// TwinCAT 3 PLC project Fraktal_Press_Demo
// Title: Fraktal_Press_Demo
// Company: fraktal-automation
// Author: fraktal-automation
// ProjectVersion: 0.1.0.10
// Description: CX2030 virtual/physical commissioning example: XTI-linked EK1200/EL1809/EL2809 HAL mapping, two-hand start, interlocked door/part slide, safety aliases, Control On/Off, AUTO/HOME/MANUAL, and model recipes.
// ProgramVersion: 3.1.4026.24
// libraries:
//   Fraktal_Core, 0.3.0.0 (fraktal-automation)
//   Fraktal_Modules, 0.2.0.0 (fraktal-automation)
//   Tc2_EtherCAT, * (Beckhoff Automation GmbH)
//   Tc2_Standard, * (Beckhoff Automation GmbH)
//   Tc2_System, * (Beckhoff Automation GmbH)
//   Tc3_Module, * (Beckhoff Automation GmbH)
// project tree:
//   00_System/Hardware/ GVL_PressIO.TcGVL (not stored), GVL_PressSafety.TcGVL (not stored)
//   00_System/ GVL_PressCommissioning.TcGVL, MAIN.TcPOU, FB_PressIoDriver.TcPOU (not stored), FB_PressControlOnCircuit.TcPOU, FB_PressControlDomain.TcPOU (not stored), FB_PressOutputAuthority.TcPOU (not stored), FB_PressSimulationDriver.TcPOU (not stored)
//   / PlcTask.TcTTO (not stored)
//   01_PneumaticPress/Sequences/ FB_PressDemoLoadPosition.TcPOU (not stored), FB_PressDemoHome.TcPOU (not stored), FB_PressDemoChangeover.TcPOU (not stored), FB_PressDemoAuto.TcPOU
//   01_PneumaticPress/Release/ FB_PressDemoRelease.TcPOU (not stored)
//   01_PneumaticPress/ FB_PressDemoUnit.TcPOU
//   01_PneumaticPress/Recipes/ FB_PressRecipeCatalog.TcPOU (not stored)
//   01_PneumaticPress/Io/ FB_PressIoCatalog.TcPOU (not stored), GVL_PressFieldbus.TcGVL (not stored)
// real-time tasks:
//   TASK PlcTask: cycle T#10ms, priority 20, ADS port 350
// I/O:
//   DEVICE =000+S-A610-A1 (EtherCAT)
// variable links:
//   Fraktal_Press_Demo/Fraktal_Press_Demo Instance <-> =000+S-A610-A1 (EtherCAT)/=000+S-K010 (EK1200)/=000+S-K010B1 (EL1809)
//     PlcTask Inputs/GVL_PressIO._000K910A <-> Channel 15/_000K910A
//     PlcTask Inputs/GVL_PressIO._000K911_Y32 <-> Channel 14/_000K911_Y32
//     PlcTask Inputs/GVL_PressIO._000MB085A_2 <-> Channel 10/_000MB085A_2
//     PlcTask Inputs/GVL_PressIO._000MB085A_4 <-> Channel 11/_000MB085A_4
//     PlcTask Inputs/GVL_PressIO._101B201A <-> Channel 3/_101B201A
//     PlcTask Inputs/GVL_PressIO._101B202A <-> Channel 5/_101B202A
//     PlcTask Inputs/GVL_PressIO._101B301A <-> Channel 1/_101B301A
//     PlcTask Inputs/GVL_PressIO._101B201B <-> Channel 4/_101B201B
//     PlcTask Inputs/GVL_PressIO._101B202B <-> Channel 6/_101B202B
//     PlcTask Inputs/GVL_PressIO._101B301B <-> Channel 2/_101B301B
//     PlcTask Inputs/GVL_PressIO._101B601 <-> Channel 12/_101B601
//     PlcTask Inputs/GVL_PressIO._101S101 <-> Channel 7/_101S101
//     PlcTask Inputs/GVL_PressIO._101S102 <-> Channel 8/_101S102
//   Fraktal_Press_Demo/Fraktal_Press_Demo Instance <-> =000+S-A610-A1 (EtherCAT)/=000+S-K010 (EK1200)/=000+S-K010C1 (EL2809)
//     PlcTask Outputs/GVL_PressIO._000K911_A1 <-> Channel 11/_000K911_A1
//     PlcTask Outputs/GVL_PressIO._000K951_A1 <-> Channel 10/_000K951_A1
//     PlcTask Outputs/GVL_PressIO._101K201A <-> Channel 3/_101K201A
//     PlcTask Outputs/GVL_PressIO._101K202A <-> Channel 5/_101K202A
//     PlcTask Outputs/GVL_PressIO._101K301A <-> Channel 1/_101K301A
//     PlcTask Outputs/GVL_PressIO._101K201B <-> Channel 4/_101K201B
//     PlcTask Outputs/GVL_PressIO._101K202B <-> Channel 6/_101K202B
//     PlcTask Outputs/GVL_PressIO._101K301B <-> Channel 2/_101K301B
//     PlcTask Outputs/GVL_PressIO._101P101 <-> Channel 7/_101P101
//     PlcTask Outputs/GVL_PressIO._101P102 <-> Channel 8/_101P102

// ---- 00_System/GVL_PressCommissioning.TcGVL
{attribute 'qualified_only'}
// Deployment-owned access-provider bootstrap. Secrets deliberately have no
// source default and are excluded from OPC UA; provision the retained values in
// the target's controlled commissioning workflow before locking the PLC policy.
VAR_GLOBAL PERSISTENT
    {attribute 'OPC.UA.DA' := '0'}
    OperatorPin   : STRING(32);
    {attribute 'OPC.UA.DA' := '0'}
    TechnicianPin : STRING(32);
    {attribute 'OPC.UA.DA' := '0'}
    AdminPin      : STRING(32);
END_VAR

// ---- 01_PneumaticPress/Sequences/FB_PressDemoAuto.TcPOU
// AUTO mode chain (Core §6.2/§6.8 ST skeleton on FB_SequenceBase): the continuous
// production cycle — await a fresh two-hand start with part+air present, transfer
// the part in, press for the recipe dwell, return to load position, count the good
// part, and loop until Stop. A Stop requested at the between-cycles wait is honored
// there (M_StopNow) so no phantom cycle is charged. Every child motion goes through
// the §6.1 handshake (M_MayIssue); progression rides the shared _retVal.
FUNCTION_BLOCK FB_PressDemoAuto EXTENDS FB_SequenceBase
VAR
    _partReady, _airReady, _startReady : BOOL;
    _dwellTwoHandHeld : BOOL;          // N220 named wait: two-hand held through the dwell
    _traceAccepted, _recordAccepted, _partProcessed : BOOL;
    {attribute 'OPC.UA.DA' := '0'}
    _pressRam : REFERENCE TO FB_CylinderCM;
    {attribute 'OPC.UA.DA' := '0'}
    _door : REFERENCE TO FB_CylinderCM;
    {attribute 'OPC.UA.DA' := '0'}
    _partSlide : REFERENCE TO FB_CylinderCM;
    {attribute 'OPC.UA.DA' := '0'}
    _twoHand : REFERENCE TO FB_TwoHandStartCM;
    {attribute 'OPC.UA.DA' := '0'}
    _partPresentSensor : REFERENCE TO FB_DigitalInputCM;
    {attribute 'OPC.UA.DA' := '0'}
    _airPressureMonitor : REFERENCE TO FB_AirPressureMonitorCM;
    {attribute 'OPC.UA.DA' := '0'}
    _parCfg : REFERENCE TO ST_PneumaticPressParCfg;
    {attribute 'OPC.UA.DA' := '0'}
    _outCmd : REFERENCE TO ST_PneumaticPressOutCmd;
    {attribute 'OPC.UA.DA' := '0'}
    _startLatched : REFERENCE TO BOOL;
    {attribute 'OPC.UA.DA' := '0'}
    _loadPosition : FB_PressDemoLoadPosition;
    _loadPositionRunning : BOOL;
END_VAR

METHOD M_Reset
M_ResetBase(0);
_loadPositionRunning := FALSE;
_loadPosition.M_Reset(BaseStepNo := 0);
END_METHOD

METHOD M_Run
IF NOT _attached THEN
    RETURN;
END_IF
CASE _step OF
    0:  // initialize
        M_Step(StepNo := 0, StepName := 'project.step.pressAutoInitialize',
            Awaits := 0, AwaitingLabel := '', TimeClass := E_TimeClass.WORK, ExpectedTime := T#0S);
        _outCmd.CycleCompleted := FALSE;
        _outCmd.Homed := FALSE;
        _outCmd.ChangeoverCompleted := FALSE;
        _loadPositionRunning := FALSE;
        _retVal := E_StepResult.ADVANCE;
        M_Advance(OnAdvance := 100, OnJump1 := -1, OnJump2 := -1, OnJump3 := -1);
    100:  // await a fresh two-hand start (the §8.11.1 cycle-start marker)
        M_Step(StepNo := 100, StepName := 'project.step.pressAwaitTwoHand',
            Awaits := 0, AwaitingLabel := '', TimeClass := E_TimeClass.WAIT_OPERATOR, ExpectedTime := T#0S);
        _outCmd.CycleCompleted := FALSE;
        _partReady := M_Await(Idx := 1, Label := 'project.condition.partPresent',
            Ok := _partPresentSensor.OutImm.Value AND _partPresentSensor.OutImm.Quality);
        _airReady := M_Await(Idx := 2, Label := 'project.condition.airPressureOk',
            Ok := _airPressureMonitor.OutImm.PressureOk);
        IF _parCfg.RequireTwoHandStart THEN
            _startReady := M_Await(Idx := 3, Label := 'project.condition.twoHandStart', Ok := _startLatched);
        ELSE
            _startReady := TRUE;
        END_IF
        IF M_StopPending() THEN
            M_StopNow();                       // stop accepted BETWEEN cycles: no phantom cycle
        ELSIF _partReady AND _airReady AND _startReady THEN
            _traceAccepted := M_PartReceived();
            _retVal := E_StepResult.ADVANCE;
        END_IF
        M_Advance(OnAdvance := 110, OnJump1 := -1, OnJump2 := -1, OnJump3 := -1);
    110:  // ram up
        M_Step(StepNo := 110, StepName := 'project.step.pressRamUp',
            Awaits := _pressRam, AwaitingLabel := 'PressRam.RETRACT', TimeClass := E_TimeClass.WORK, ExpectedTime := T#0S);
        IF M_MayIssue(Steppable := TRUE) THEN
            _pressRam.Abort := FALSE; _pressRam.Command := E_CylinderCommand.RETRACT; _pressRam.Execute := TRUE;
        END_IF
        IF _pressRam.Done THEN _pressRam.Execute := FALSE; _retVal := E_StepResult.ADVANCE; END_IF
        M_Advance(OnAdvance := 130, OnJump1 := -1, OnJump2 := -1, OnJump3 := -1);
    130:  // door open
        M_Step(StepNo := 130, StepName := 'project.step.pressDoorOpen',
            Awaits := _door, AwaitingLabel := 'Door.RETRACT', TimeClass := E_TimeClass.WORK, ExpectedTime := T#0S);
        IF M_MayIssue(Steppable := TRUE) THEN
            _door.Abort := FALSE; _door.Command := E_CylinderCommand.RETRACT; _door.Execute := TRUE;
        END_IF
        IF _door.Done THEN _door.Execute := FALSE; _retVal := E_StepResult.ADVANCE; END_IF
        M_Advance(OnAdvance := 150, OnJump1 := -1, OnJump2 := -1, OnJump3 := -1);
    150:  // slide inside (value-adding sequence begins)
        M_Step(StepNo := 150, StepName := 'project.step.pressSlideInside',
            Awaits := _partSlide, AwaitingLabel := 'PartSlide.EXTEND', TimeClass := E_TimeClass.WORK, ExpectedTime := T#0S);
        IF M_MayIssue(Steppable := TRUE) THEN
            M_PartStarted();
            _partSlide.Abort := FALSE; _partSlide.Command := E_CylinderCommand.EXTEND; _partSlide.Execute := TRUE;
        END_IF
        IF _partSlide.Done THEN _partSlide.Execute := FALSE; _retVal := E_StepResult.ADVANCE; END_IF
        M_Advance(OnAdvance := 170, OnJump1 := -1, OnJump2 := -1, OnJump3 := -1);
    170:  // transfer settle
        M_Step(StepNo := 170, StepName := 'project.step.pressTransferSettle',
            Awaits := 0, AwaitingLabel := '', TimeClass := E_TimeClass.WORK, ExpectedTime := _parCfg.TransferSettleTime);
        _retVal := M_Delay(PT := _parCfg.TransferSettleTime);
        M_Advance(OnAdvance := 180, OnJump1 := -1, OnJump2 := -1, OnJump3 := -1);
    180:  // door close
        M_Step(StepNo := 180, StepName := 'project.step.pressDoorClose',
            Awaits := _door, AwaitingLabel := 'Door.EXTEND', TimeClass := E_TimeClass.WORK, ExpectedTime := T#0S);
        IF M_MayIssue(Steppable := TRUE) THEN
            _door.Abort := FALSE; _door.Command := E_CylinderCommand.EXTEND; _door.Execute := TRUE;
        END_IF
        IF _door.Done THEN _door.Execute := FALSE; _retVal := E_StepResult.ADVANCE; END_IF
        M_Advance(OnAdvance := 200, OnJump1 := -1, OnJump2 := -1, OnJump3 := -1);
    200:  // ram down
        M_Step(StepNo := 200, StepName := 'project.step.pressRamDown',
            Awaits := _pressRam, AwaitingLabel := 'PressRam.EXTEND', TimeClass := E_TimeClass.WORK, ExpectedTime := T#0S);
        IF M_MayIssue(Steppable := TRUE) THEN
            _pressRam.Abort := FALSE; _pressRam.Command := E_CylinderCommand.EXTEND; _pressRam.Execute := TRUE;
        END_IF
        IF _pressRam.Done THEN _pressRam.Execute := FALSE; _retVal := E_StepResult.ADVANCE; END_IF
        M_Advance(OnAdvance := 220, OnJump1 := -1, OnJump2 := -1, OnJump3 := -1);
    220:  // press dwell — two-hand must stay held; releasing it HOLDS the dwell
        M_Step(StepNo := 220, StepName := 'project.step.pressDwell',
            Awaits := 0, AwaitingLabel := '', TimeClass := E_TimeClass.WORK, ExpectedTime := _parCfg.PressSettleTime);
        // Releasing the button mid-dwell is the designed way to stop pressing, so it
        // is a named wait (§6.9(b)), not a fault: the ram's outputs come off, the
        // dwell timer freezes where it is because M_Delay is not called, and pressing
        // again restores the force and finishes the remaining dwell. Faulting here
        // charged an unrecoverable downtime event for normal operator behaviour.
        _dwellTwoHandHeld := M_Await(Idx := 1, Label := 'project.condition.twoHandHeldDuringPress',
            Ok := _twoHand.OutImm.SafeActive OR NOT _parCfg.RequireTwoHandStart);
        IF NOT _dwellTwoHandHeld THEN
            _pressRam.WithdrawOutputs();
        ELSE
            // The press force is the valve latched by the EXTEND that step 200 already
            // completed, so after a withdraw only this call re-energizes it — and the
            // ram re-checks its own extend permit before it does (§7.2).
            _pressRam.RestoreOutputs();
            _retVal := M_Delay(PT := _parCfg.PressSettleTime);
        END_IF
        M_Advance(OnAdvance := 230, OnJump1 := -1, OnJump2 := -1, OnJump3 := -1);
    230:  // record the applied dwell (§3.16.1 measured value)
        M_Step(StepNo := 230, StepName := 'project.step.pressRecordResult',
            Awaits := 0, AwaitingLabel := '', TimeClass := E_TimeClass.WORK, ExpectedTime := T#0S);
        _recordAccepted := M_PartRecord(RecordName := 'PressDwell',
            Value := DINT_TO_LREAL(TIME_TO_DINT(_parCfg.PressSettleTime)),
            Minimum := 0, Maximum := 30000,
            Target := DINT_TO_LREAL(TIME_TO_DINT(_parCfg.PressSettleTime)), EngUnit := 'ms');
        _loadPositionRunning := FALSE;
        _retVal := E_StepResult.ADVANCE;
        M_Advance(OnAdvance := 240, OnJump1 := -1, OnJump2 := -1, OnJump3 := -1);
    240:  // return to the shared load-safe position (composite step)
        IF NOT _loadPositionRunning THEN
            _loadPosition.M_Reset(BaseStepNo := 240);
            _loadPositionRunning := TRUE;
        END_IF
        _loadPosition.M_Run();
        IF _loadPosition.Done THEN
            _loadPositionRunning := FALSE;
            _retVal := E_StepResult.ADVANCE;
        END_IF
        M_Advance(OnAdvance := 999, OnJump1 := -1, OnJump2 := -1, OnJump3 := -1);
    999:  // cycle complete — write result, count by verdict, loop (§8.11.1 finish marker)
        M_Step(StepNo := 999, StepName := 'project.step.pressAutoComplete',
            Awaits := 0, AwaitingLabel := '', TimeClass := E_TimeClass.WORK, ExpectedTime := T#0S);
        _outCmd.CycleCompleted := TRUE;
        _partProcessed := M_PartProcessed(Verdict := E_Verdict.OK, Reason := E_Reason.NONE);
        IF NOT _partProcessed THEN
            M_CountGood();                     // §3.9: no carrier configured — count directly
        END_IF
        _startLatched := FALSE;
        IF M_EndOfCycle() THEN
            _retVal := E_StepResult.ADVANCE;   // stop NOT requested: loop to N100
        END_IF
        M_Advance(OnAdvance := 100, OnJump1 := -1, OnJump2 := -1, OnJump3 := -1);
ELSE
    M_Fault(Reason := E_Reason.STEP_STALLED, DescriptionKey := 'std.error.undefinedStep');
END_CASE
END_METHOD

METHOD Setup : BOOL
VAR_INPUT
    Host : I_SequenceHost;
END_VAR
VAR_IN_OUT
    PressRam : FB_CylinderCM;
    Door : FB_CylinderCM;
    PartSlide : FB_CylinderCM;
    TwoHand : FB_TwoHandStartCM;
    PartPresentSensor : FB_DigitalInputCM;
    AirPressureMonitor : FB_AirPressureMonitorCM;
    ParCfg : ST_PneumaticPressParCfg;
    OutCmd : ST_PneumaticPressOutCmd;
    StartLatched : BOOL;
END_VAR
_pressRam REF= PressRam;
_door REF= Door;
_partSlide REF= PartSlide;
_twoHand REF= TwoHand;
_partPresentSensor REF= PartPresentSensor;
_airPressureMonitor REF= AirPressureMonitor;
_parCfg REF= ParCfg;
_outCmd REF= OutCmd;
_startLatched REF= StartLatched;
Setup := M_Attach(Host := Host) AND __ISVALIDREF(_pressRam) AND __ISVALIDREF(_door)
    AND __ISVALIDREF(_partSlide) AND __ISVALIDREF(_twoHand)
    AND __ISVALIDREF(_partPresentSensor) AND __ISVALIDREF(_airPressureMonitor)
    AND __ISVALIDREF(_parCfg) AND __ISVALIDREF(_outCmd) AND __ISVALIDREF(_startLatched)
    AND _loadPosition.Setup(Host := Host, PressRam := PressRam, Door := Door, PartSlide := PartSlide);
END_METHOD

END_FUNCTION_BLOCK

// ---- 01_PneumaticPress/FB_PressDemoUnit.TcPOU
// Project-owned Unit: pneumatic press + access door + transfer slide + two-hand request.
// Cylinder interlocks prevent the two documented collisions in AUTO and MANUAL.
// Certified E-stop, two-hand evaluation and safe valve outputs remain external.
FUNCTION_BLOCK FB_PressDemoUnit EXTENDS FB_UnitBase
VAR_INPUT
    ParCfg : ST_PneumaticPressParCfg;
    ParCmd : ST_PneumaticPressParCmd;
END_VAR
VAR_OUTPUT
    PressRam      : FB_CylinderCM;
    Door          : FB_CylinderCM;
    PartSlide     : FB_CylinderCM;
    TwoHand       : FB_TwoHandStartCM;
    PneumaticPower: FB_PowerGroupCM;
    PartPresentSensor : FB_DigitalInputCM;
    AirPressureMonitor : FB_AirPressureMonitorCM;
    ReleaseConditions : FB_PressDemoRelease; // project-owned, browseable condition state
    OutCmd        : ST_PneumaticPressOutCmd;
    OutImm        : ST_PneumaticPressOutImm;
END_VAR
VAR
    {attribute 'OPC.UA.DA' := '0'}
    _recipe : I_RecipeProvider;
    _parCfgStaged : ST_PneumaticPressParCfg;
    _recipePrepared : BOOL;
    _startLatched : BOOL;
    _powerRequestPending : BOOL;
    _powerTargetOn : BOOL;
    {attribute 'OPC.UA.DA' := '0'}
    _homeSequence : FB_PressDemoHome;       // §6.8 ST chain on FB_SequenceBase owns HOME steps
    {attribute 'OPC.UA.DA' := '0'}
    _changeoverSequence : FB_PressDemoChangeover;
    {attribute 'OPC.UA.DA' := '0'}
    _autoSequence : FB_PressDemoAuto;
END_VAR

Cyclic();

METHOD Setup : BOOL
VAR_INPUT
    Name : STRING(80);
    PressHal : REFERENCE TO ST_CylinderHal;
    DoorHal : REFERENCE TO ST_CylinderHal;
    SlideHal : REFERENCE TO ST_CylinderHal;
    TwoHandHal : REFERENCE TO ST_TwoHandHal;
    PowerHal : REFERENCE TO ST_PowerGroupHal;
    PartPresentHal : REFERENCE TO ST_DigitalInputHal;
    AirPressureHal : REFERENCE TO ST_AirPressureHal;
    Recipe : I_RecipeProvider;
END_VAR
VAR
    InitialModel : ST_ModelId;
    Ok : BOOL;
END_VAR
_M_SetName(Name);
_M_SetPresentation(DisplayNameKey := 'project.module.pneumaticPress.name', DescriptionKey := 'project.module.pneumaticPress.description');
_recipe := Recipe;
Ok := PressRam.Setup(Name := CONCAT(Name, '.PressRam'), HalRef := PressHal, Recipe := 0);
Ok := Door.Setup(Name := CONCAT(Name, '.Door'), HalRef := DoorHal, Recipe := 0) AND Ok;
Ok := PartSlide.Setup(Name := CONCAT(Name, '.PartSlide'), HalRef := SlideHal, Recipe := 0) AND Ok;
Ok := TwoHand.Setup(Name := CONCAT(Name, '.TwoHand'), HalRef := TwoHandHal) AND Ok;
Ok := PneumaticPower.Setup(Name := CONCAT(Name, '.PneumaticPower'), HalRef := PowerHal) AND Ok;
Ok := PartPresentSensor.Setup(Name := CONCAT(Name, '.PartPresentSensor'),
    HalRef := PartPresentHal, DisplayNameKey := 'project.module.partPresentSensor.name',
    DescriptionKey := 'project.module.partPresentSensor.description') AND Ok;
Ok := AirPressureMonitor.Setup(Name := CONCAT(Name, '.AirPressureMonitor'),
    HalRef := AirPressureHal) AND Ok;
Ok := ReleaseConditions.Setup(UnitPath := Name) AND Ok;
Ok := _homeSequence.Setup(Host := THIS^, PressRam := PressRam, Door := Door,
    PartSlide := PartSlide, OutCmd := OutCmd) AND Ok;
Ok := _changeoverSequence.Setup(Host := THIS^, PressRam := PressRam, Door := Door,
    PartSlide := PartSlide, OutCmd := OutCmd, Model := Model) AND Ok;
Ok := _autoSequence.Setup(Host := THIS^, PressRam := PressRam, Door := Door,
    PartSlide := PartSlide, TwoHand := TwoHand, PartPresentSensor := PartPresentSensor,
    AirPressureMonitor := AirPressureMonitor, ParCfg := ParCfg, OutCmd := OutCmd,
    StartLatched := _startLatched) AND Ok;
PneumaticPower.ParCfg.Kind := E_PowerGroupKind.VALVE_ZONE;
PneumaticPower.ParCfg.RequiredForControl := TRUE;
PneumaticPower.ParCfg.FieldbusLossReaction := E_FieldbusLossReaction.CONTROL_OFF;
Ok := _M_Register(PressRam) AND Ok;
Ok := _M_Register(Door) AND Ok;
Ok := _M_Register(PartSlide) AND Ok;
Ok := _M_Register(TwoHand) AND Ok;
Ok := _M_Register(PneumaticPower) AND Ok;
Ok := _M_Register(PartPresentSensor) AND Ok;
Ok := _M_Register(AirPressureMonitor) AND Ok;
Setup := Ok AND PrepareRecipe(Model := InitialModel);
IF Setup THEN CommitRecipe(); END_IF
END_METHOD

METHOD PrepareRecipe : BOOL
VAR_INPUT
    Model : ST_ModelId;
END_VAR
IF _recipe = 0 THEN
    _parCfgStaged := ParCfg;
    _recipePrepared := TRUE;
ELSIF _recipe.Load(ModelCode := Model.ModelCode, RecipeKey := 'PneumaticPressUnit', pParCfg := ADR(_parCfgStaged), Size := SIZEOF(_parCfgStaged)) THEN
    IF (_parCfgStaged.PressSettleTime > T#30S) OR (_parCfgStaged.TransferSettleTime > T#5S) THEN
        _M_Fault(E_Reason.RECIPE_INVALID, 'project.error.pressRecipeInvalid');
        _recipePrepared := FALSE;
        PrepareRecipe := FALSE;
        RETURN;
    END_IF
    _recipePrepared := TRUE;
ELSE
    _M_Fault(E_Reason.RECIPE_INVALID, 'std.error.recipeSchemaInvalid');
    _recipePrepared := FALSE;
    PrepareRecipe := FALSE;
    RETURN;
END_IF
PrepareRecipe := SUPER^.PrepareRecipe(Model := Model);
IF NOT PrepareRecipe THEN _recipePrepared := FALSE; END_IF
END_METHOD

METHOD CommitRecipe
SUPER^.CommitRecipe();
IF _recipePrepared THEN
    ParCfg := _parCfgStaged;
    // §8.11 performance references follow the model: OEE Performance denominator
    // and the WORK-time degradation baseline are per-recipe engineering data.
    Oee.IdealCycleMs := ParCfg.IdealCycleMs;
    Profiler.M_SetBaselineWork(WorkMs := ParCfg.BaselineWorkMs);
END_IF
_recipePrepared := FALSE;
END_METHOD

METHOD AbortRecipe
SUPER^.AbortRecipe();
_recipePrepared := FALSE;
END_METHOD

// First operational scan: initialize application-owned mode-chain state.
METHOD PROTECTED OnInit : DINT
OnInit := SUPER^.OnInit();
_M_ResetModeSequences();
_M_ClearModeTransitionState();
END_METHOD

// Every accepted Unit Start gets a fresh mode chain, including a repeated
// HOME/CHANGEOVER run that does not pass through another mode change.
METHOD PROTECTED OnCommandStart : DINT
OnCommandStart := SUPER^.OnCommandStart();
_M_ResetModeSequences();
END_METHOD

// Mode-entry wiring only. Step behavior remains in the selected sequence POU.
METHOD PROTECTED OnModeChanged : DINT
VAR_INPUT
    NewMode : E_Mode;
    OldMode : E_Mode;
END_VAR
OnModeChanged := SUPER^.OnModeChanged(
    NewMode := NewMode, OldMode := OldMode);
_M_ResetModeSequences();
_M_ClearModeTransitionState();
END_METHOD

METHOD PROTECTED OnCyclic : DINT
OnCyclic := SUPER^.OnCyclic();
// Project release engineering is a separate visible component. It owns the
// functional collision permits and mode-entry conditions consumed below.
ReleaseConditions.M_Evaluate(PressRam := PressRam, Door := Door, PartSlide := PartSlide,
    TwoHand := TwoHand, PneumaticPower := PneumaticPower,
    AirPressure := AirPressureMonitor);

// Latch access-gated Unit requests, then observe one full Execute-low scan before
// starting another power-group command (PLCopen edge discipline).
IF ControlOffRequest THEN
    _powerTargetOn := FALSE;
    _powerRequestPending := TRUE;
ELSIF ControlOnRequest THEN
    _powerTargetOn := TRUE;
    _powerRequestPending := TRUE;
END_IF
IF PneumaticPower.Done OR PneumaticPower.Error OR PneumaticPower.Aborted THEN
    PneumaticPower.Execute := FALSE;
ELSIF _powerRequestPending AND NOT PneumaticPower.Execute
AND (PneumaticPower.State = E_ExecState.READY) THEN
    PneumaticPower.Abort := FALSE;
    IF _powerTargetOn THEN
        PneumaticPower.Command := E_PowerGroupCommand.POWER_ON;
    ELSE
        PneumaticPower.Command := E_PowerGroupCommand.POWER_OFF;
    END_IF
    PneumaticPower.Execute := TRUE;
    _powerRequestPending := FALSE;
END_IF

// A physical two-hand edge may start AUTO from READY, or release an already
// running Unit's wait step. It never bypasses domain readiness or access policy.
IF TwoHand.OutImm.StartPulse
AND PartPresentSensor.OutImm.Value AND PartPresentSensor.OutImm.Quality
AND AirPressureMonitor.OutImm.PressureOk THEN
    IF (State = E_ExecState.BUSY) AND (ModeActive = E_Mode.AUTO) THEN
        _startLatched := TRUE;
    ELSIF (ModeActive = E_Mode.AUTO) AND Start() THEN
        _startLatched := TRUE;
    END_IF
ELSIF TwoHand.OutImm.StartPulse THEN
    _startLatched := FALSE;
END_IF
IF PneumaticPower.Error AND (State = E_ExecState.BUSY) THEN
    _M_RollupFault();
END_IF
IF (State = E_ExecState.BUSY)
AND NOT AirPressureMonitor.OutImm.PressureOk THEN
    PressRam.WithdrawOutputs();
    Door.WithdrawOutputs();
    PartSlide.WithdrawOutputs();
    _M_Fault(E_Reason.PERMISSIVE_NOT_MET, 'project.error.pressAirPressureLost');
END_IF
OutImm.PressRetracted := PressRam.OutImm.Retracted;
OutImm.DoorOpen := Door.OutImm.Retracted;
OutImm.DoorClosed := Door.OutImm.Extended;
OutImm.SlideInside := PartSlide.OutImm.Extended;
OutImm.SlideOutside := PartSlide.OutImm.Retracted;
OutImm.TwoHandArmed := TwoHand.OutImm.Armed;
OutImm.TwoHandActive := TwoHand.OutImm.SafeActive;
OutImm.PartPresent := PartPresentSensor.OutImm.Value AND PartPresentSensor.OutImm.Quality;
OutImm.AirPressureOk := AirPressureMonitor.OutImm.PressureOk;
OutImm.ReadyForLoad := Door.OutImm.Retracted AND NOT Door.OutImm.Extended
    AND PartSlide.OutImm.Retracted AND NOT PartSlide.OutImm.Extended
    AND PressRam.OutImm.Retracted AND NOT PressRam.OutImm.Extended;
OutImm.ActiveSettleTime := ParCfg.PressSettleTime;
OutImm.Diagnostic := Status.Diagnostic;
END_METHOD

METHOD PROTECTED OnAbort : DINT
OnAbort := SUPER^.OnAbort();
_M_PartAborted();                    // §3.16.3: the part leaves without a valid result
_M_WithdrawSequenceOutputs();
_M_ResetModeSequences();
_M_ClearModeTransitionState();
_powerTargetOn := FALSE;
_powerRequestPending := TRUE;
END_METHOD

// Error-state Abort is a deliberate recovery action but does not clear ERROR.
METHOD PROTECTED OnAbortInError : DINT
OnAbortInError := SUPER^.OnAbortInError();
_M_WithdrawSequenceOutputs();
_M_ResetModeSequences();
_M_ClearModeTransitionState();
_powerTargetOn := FALSE;
_powerRequestPending := TRUE;
END_METHOD

// An operator reset is recovering this Unit: put the application back to the same
// safe wiring an error-state abort establishes, so the reset the operator presses at
// the panel needs no separate Stop/Abort first. The base then releases the run
// command and the children's commands, so the next HOME gets a genuine command edge.
// Unlike the abort paths this does NOT touch control power in either direction: it
// never requests Control On (§9.8 forbids self-resume), and it must not request
// Control Off either — powering down a healthy control circuit would make the
// operator re-enable it before HOME could run, i.e. reintroduce the multi-action
// recovery this reset exists to remove. Power stays where the operator put it.
METHOD PROTECTED OnOperatorReset : DINT
OnOperatorReset := SUPER^.OnOperatorReset();
_M_WithdrawSequenceOutputs();
_M_ResetModeSequences();
_M_ClearModeTransitionState();
END_METHOD

// One safe-stop wiring point shared by normal and error-state abort transitions.
METHOD PROTECTED _M_WithdrawSequenceOutputs
PressRam.WithdrawOutputs();
Door.WithdrawOutputs();
PartSlide.WithdrawOutputs();
PressRam.Execute := FALSE;
Door.Execute := FALSE;
PartSlide.Execute := FALSE;
END_METHOD

// Reset application-owned chain plumbing at lifecycle transitions. The chains'
// N000/N999 steps remain the only owners of process initialization/completion.
METHOD PROTECTED _M_ResetModeSequences
_homeSequence.M_Reset();
_changeoverSequence.M_Reset();
_autoSequence.M_Reset();
END_METHOD

// Clear state that must not survive init, mode entry, or either abort path.
// OnCommandStart deliberately does not call this: a physical start pulse may have
// been latched one scan before the inherited Execute edge is consumed.
METHOD PROTECTED _M_ClearModeTransitionState
Decision.Prompt := '';
DecisionAnswer := 0;
_startLatched := FALSE;
END_METHOD

// Application-only seam for ordinary hardwired Control On/Off buttons.
// It is a method (not OPC UA data), so HMI writes still use the access-gated
// ReqControlOn/ReqControlOff contract. The power CM rechecks safety and health.
METHOD RequestLocalControl : BOOL
VAR_INPUT
    ControlOn : BOOL;
END_VAR
_powerTargetOn := ControlOn;
_powerRequestPending := TRUE;
RequestLocalControl := TRUE;
END_METHOD

// §3.4.2 — the press paces every motion boundary through _M_StepGate, so
// SINGLE_STEP and HOLD_TO_RUN are supported (NON-SAFETY pacing; interlocks
// and the certified safety layer are unaffected).
METHOD PROTECTED _M_SupportsRunStyle : BOOL
VAR_INPUT
    Style : E_RunStyle;
END_VAR
_M_SupportsRunStyle := (Style = E_RunStyle.CONTINUOUS)
    OR (Style = E_RunStyle.SINGLE_STEP) OR (Style = E_RunStyle.HOLD_TO_RUN);
END_METHOD

METHOD PROTECTED _M_Supports : BOOL
VAR_INPUT
    Mode : E_Mode;
END_VAR
_M_Supports := (Mode = E_Mode.AUTO) OR (Mode = E_Mode.MANUAL)
    OR (Mode = E_Mode.HOME) OR (Mode = E_Mode.CHANGEOVER);
END_METHOD

// Thin mode router. Each supported sequence is a named method in the Unit tree.
METHOD PROTECTED _M_Dispatch
CASE ModeActive OF
    E_Mode.AUTO:
        _M_SequenceAuto();
    E_Mode.HOME:
        _M_SequenceHome();
    E_Mode.CHANGEOVER:
        _M_SequenceChangeover();
    E_Mode.MANUAL:
        _M_Fault(E_Reason.UNSUPPORTED_COMMAND, 'project.error.pressManualHasNoSequence');
ELSE
    _M_Fault(E_Reason.UNSUPPORTED_COMMAND, 'project.error.pressModeHasNoSequence');
END_CASE
END_METHOD

// Wiring-only HOME adapter. OnCommandStart owns the reset edge; the sequence POU
// owns every process step and terminal action.
METHOD PROTECTED _M_SequenceHome
_homeSequence.M_Run();
END_METHOD

// Wiring-only CHANGEOVER adapter. The §6.8 chain owns model validation, safe
// positioning, the operator decision, and completion logic.
METHOD PROTECTED _M_SequenceChangeover
_changeoverSequence.M_Run();
END_METHOD

// Wiring-only AUTO adapter. Every production command, wait, timer, decision,
// traceability action, and transition lives in the §6.8 chain.
METHOD PROTECTED _M_SequenceAuto
_autoSequence.M_Run();
END_METHOD

METHOD PROTECTED _M_RouteManual : BOOL
VAR_INPUT
    TargetPath : STRING(255);
    Value : DINT;
END_VAR
_M_RouteManual := FALSE;
IF TargetPath = PressRam.Name THEN
    _M_RouteManual := PressRam.ManualCommand(Value := Value);
ELSIF TargetPath = Door.Name THEN
    _M_RouteManual := Door.ManualCommand(Value := Value);
ELSIF TargetPath = PartSlide.Name THEN
    _M_RouteManual := PartSlide.ManualCommand(Value := Value);
ELSE
    _M_RouteManual := FALSE;
END_IF
END_METHOD

// §7.8 mode-entry release owned by this Unit. The base Start method consumes the
// same report the HMI displays, so this condition cannot become explanation-only.
METHOD PROTECTED _M_AppendInterlocks
VAR_IN_OUT
    Report : ST_ReleaseReport;
END_VAR
ReleaseConditions.M_AppendStart(Report := Report);
END_METHOD

METHOD PROTECTED _M_AppendManualInterlocks
VAR_INPUT
    TargetPath : STRING(255);
    Value : DINT;
END_VAR
VAR_IN_OUT
    Report : ST_ReleaseReport;
END_VAR
ReleaseConditions.M_AppendManual(TargetPath := TargetPath, Value := Value,
    PressRam := PressRam, Door := Door, PartSlide := PartSlide, Report := Report);
END_METHOD

METHOD PROTECTED _M_PublishStatus
SUPER^._M_PublishStatus();
OutImm.Diagnostic := Status.Diagnostic;
END_METHOD

// §3.10.2 — base walk (Unit facets + all child modules), then the project-owned
// fieldbus topology identity: static members of GVL_PressFieldbus.Topology are
// OPC.UA.DA=0 and reach the HMI only through this manifest.
METHOD M_AppendConfig : BOOL
VAR_INPUT
    Pager : REFERENCE TO FB_ConfigPager;
END_VAR
M_AppendConfig := SUPER^.M_AppendConfig(Pager := Pager);
F_AppendTopologyConfig(Topology := GVL_PressFieldbus.Topology, Pager := Pager);
END_METHOD

END_FUNCTION_BLOCK

// ---- 00_System/MAIN.TcPOU
// Virtual-commissioning application for one pneumatic press Unit.
// IMPORTANT: the Safe* values below simulate TwinSAFE outputs only. A deployed
// machine maps certified E-stop/two-hand/guard/safe-valve results from TwinSAFE.
PROGRAM MAIN
VAR
    RecipeCatalog : FB_PressRecipeCatalog;
    PartCarrier : FB_LocalPartCarrier;    // §3.16.2 BY_POSITION identity + local result ring
    AccessUsers : FB_LocalAccessProvider; // §7.7 commissioning user/PIN table
    // TF6100 TMC-Filtered publication starts at the deployed root instance.
    // The marker is inherited by PneumaticPress's published child symbols.
    {attribute 'OPC.UA.DA' := '1'}
    PneumaticPress : FB_PressDemoUnit;
    IoCatalog : FB_PressIoCatalog;
    IoDriver : FB_PressIoDriver;
    ControlDomain : FB_PressControlDomain;
    OutputAuthority : FB_PressOutputAuthority;
    SimulationDriver : FB_PressSimulationDriver;
    PressHal, DoorHal, SlideHal : ST_CylinderHal;
    TwoHandHal : ST_TwoHandHal;
    PowerHal : ST_PowerGroupHal;
    PartPresentHal : ST_DigitalInputHal;
    AirPressureHal : ST_AirPressureHal;
    HealthProbe : FB_TcSystemHealthProbe;
    HealthConfig : ST_SystemHealthParCfg;
    HealthCpuLoadPct : LREAL;
    HealthMemoryAvailableMb : UDINT;
    HealthTimeSource : STRING(32);
    InitialModel : ST_ModelId;
    Plate : ST_Nameplate;
    Init : BOOL;
    // Read-only MIRRORS of the commissioning gates (see the VAR CONSTANT block).
    // They exist only so the gate state stays visible over ADS/OPC UA: the
    // compiler inlines constants, which may publish no symbol at all, and losing
    // that visibility would remove the fastest way to diagnose "no output moves".
    // They are reassigned from the constants every cycle and nothing reads them,
    // so writing one online is inert - the constant remains the only authority.
    UseSimulation : BOOL;
    ControlCircuitMappingConfirmed : BOOL;
    // §10.5.1 demand gate, written by the HMI while its fieldbus page is open.
    // FALSE parks the EtherCAT master scan (no ADS traffic for a view nobody is
    // watching); the last read states are held, never falsified.
    FieldbusViewActive : BOOL;

    // Simulation controls. E-stop is normally closed: TRUE = healthy circuit.
    SimEStopNc : BOOL := TRUE;
    SimControlOnButton : BOOL;
    SimControlOffButton : BOOL;
    SimLeftButton : BOOL;
    SimRightButton : BOOL;
    SimSafetyValveOk : BOOL := TRUE;
    SimFieldbusHealthy : BOOL := TRUE;
    SimPartPresent : BOOL := TRUE;
    SimAirPressureOk : BOOL := TRUE;
    SafeEStopOk : BOOL;
    SafeGuardClosed : BOOL;
    SafeTwoHandActive : BOOL;
    SafePneumaticPermit : BOOL;
    SafetyFieldbusHealthy : BOOL;
    StandardIoHealthy : BOOL;
    RawEStopHealthy : BOOL;
    LampsOn : BOOL;
    ControlOnEdge : R_TRIG;
    ControlOffEdge : R_TRIG;
    ControlOnAdopted : R_TRIG;   // rising edge of the relay chain's feedback
END_VAR
VAR CONSTANT
    // COMMISSIONING GATES - deliberately CONSTANT so they cannot be flipped
    // online. Defeating a gate must be a source change plus a download: a
    // reviewable, auditable act, not a live write from an HMI or ADS client.
    //
    // TRUE makes MAIN call M_ClearOutputs() every cycle, so no physical output
    // is ever energized while the simulation driver animates the plant.
    USE_SIMULATION : BOOL := FALSE;
    // FALSE makes M_WriteOutputs force _000K951_A1 and _000K911_A1 FALSE every
    // cycle. Control On then cannot energize, the hardwired N54 D2 relay chain
    // never closes, and NOTHING moves - even though the cylinder coils are
    // written unconditionally. Set TRUE only after verifying the K951/K911
    // electrical semantics on the cabinet; per N54 D2 SwitchControlOn and
    // EnableControlOn are distinct signals.
    CONTROL_CIRCUIT_MAPPING_CONFIRMED : BOOL := TRUE;
END_VAR

// Mirror the compile-time gates so they remain observable (see declaration).
UseSimulation := USE_SIMULATION;
ControlCircuitMappingConfirmed := CONTROL_CIRCUIT_MAPPING_CONFIRMED;

IF NOT Init THEN
    Init := TRUE;
    // Initial mechanically safe/load position: ram up, door open, slide outside.
    PressHal.RetractedFb := TRUE;
    DoorHal.RetractedFb := TRUE;
    SlideHal.RetractedFb := TRUE;
    RecipeCatalog.Setup(UnitRef := PneumaticPress);
    PneumaticPress.Setup(Name := 'PneumaticPress', PressHal := PressHal, DoorHal := DoorHal,
        SlideHal := SlideHal, TwoHandHal := TwoHandHal, PowerHal := PowerHal,
        PartPresentHal := PartPresentHal, AirPressureHal := AirPressureHal,
        Recipe := RecipeCatalog.Provider);
    IoDriver.Setup(UnitRef := PneumaticPress);
    IoCatalog.Setup(UnitRef := PneumaticPress);
    ControlDomain.Setup(UnitRef := PneumaticPress);
    SimulationDriver.Setup(PressHal := PressHal, DoorHal := DoorHal, SlideHal := SlideHal);
    InitialModel.ModelCode := 'ALUMINUM';
    PneumaticPress.SetModel(Id := InitialModel);
    Plate.ProductUri := 'urn:fraktal:demo:pneumatic-press:2026-0001';
    Plate.ManufacturerName := 'Fraktal Example Project';
    Plate.ProductDesignation := 'Pneumatic Press Training Cell';
    Plate.SerialNumber := 'PRESS-DEMO-2026-0001';
    Plate.YearOfConstruction := '2026';
    Plate.SoftwareVersion := 'Fraktal Press Demo 0.1';
    PneumaticPress.SetNameplate(Plate := Plate);
    PneumaticPress.AlarmLog.RegisterMeta(Reason := E_Reason.INTERLOCK_DROPPED,
        OperatorAction := 'project.alarmAction.pressInterlock',
        Consequence := 'project.alarmConsequence.pressInterlock', Shelvable := FALSE);
    // §8.9 rationalization: per-reason operator action + consequence for the HMI join
    PneumaticPress.AlarmLog.RegisterMeta(Reason := E_Reason.PERMISSIVE_NOT_MET,
        OperatorAction := 'project.alarmAction.pressAirPressure',
        Consequence := 'project.alarmConsequence.pressAirPressure', Shelvable := FALSE);
    PneumaticPress.AlarmLog.RegisterMeta(Reason := E_Reason.RECIPE_INVALID,
        OperatorAction := 'project.alarmAction.pressRecipe',
        Consequence := 'project.alarmConsequence.pressRecipe', Shelvable := FALSE);
    PneumaticPress.AlarmLog.RegisterMeta(Reason := PL_ModuleReasons.CYL_WORK_NOT_REACHED,
        OperatorAction := 'project.alarmAction.pressCylinderPosition',
        Consequence := 'project.alarmConsequence.pressCylinderPosition', Shelvable := FALSE);
    PneumaticPress.AlarmLog.RegisterMeta(Reason := PL_ModuleReasons.CYL_HOME_NOT_REACHED,
        OperatorAction := 'project.alarmAction.pressCylinderPosition',
        Consequence := 'project.alarmConsequence.pressCylinderPosition', Shelvable := FALSE);
    // §3.16 traceability: station-local BY_POSITION serials; RFID/host substitutes later
    PartCarrier.Setup(UidPrefix := 'PRESS-2026-');
    PneumaticPress.SetPartCarrier(Carrier := PartCarrier);
    // §7.7/§14: provider secrets are retained deployment configuration, never
    // source literals. Provision them before raising any policy threshold.
    IF GVL_PressCommissioning.OperatorPin <> '' THEN
        AccessUsers.Register(User := 'operator', Pin := GVL_PressCommissioning.OperatorPin,
            Level := E_AccessLevel.OPERATOR);
    ELSE
        ;
    END_IF
    IF GVL_PressCommissioning.TechnicianPin <> '' THEN
        AccessUsers.Register(User := 'tech', Pin := GVL_PressCommissioning.TechnicianPin,
            Level := E_AccessLevel.TECHNICIAN);
    ELSE
        ;
    END_IF
    IF GVL_PressCommissioning.AdminPin <> '' THEN
        AccessUsers.Register(User := 'admin', Pin := GVL_PressCommissioning.AdminPin,
            Level := E_AccessLevel.ADMIN);
    ELSE
        ;
    END_IF
    PneumaticPress.Access.Setup(Provider := AccessUsers, pAlarmLog := ADR(PneumaticPress.AlarmLog));
    HealthConfig.MaxTaskCycleUs := 5000;
    HealthConfig.MaxTaskJitterUs := 2000;
    HealthConfig.RequireFieldbus := TRUE;
    HealthConfig.RequireDcSync := FALSE;
    HealthConfig.RequireTimeSync := TRUE;
END_IF

// Ordinary simulated local station buttons. The worksheet does not list real
// Control On/Off input buttons; physical operation therefore uses HMI requests
// until those devices are identified. Control Off wins simultaneous edges.
// Source the Control On/Off edges from the REAL buttons on a live machine, and
// from the simulated ones only under USE_SIMULATION. Previously both edges were
// ANDed with USE_SIMULATION, so on hardware neither could ever fire and the
// machine had no headless Control On path at all.
IF USE_SIMULATION THEN
    ControlOnEdge(CLK := SimControlOnButton);
    ControlOffEdge(CLK := SimControlOffButton);
ELSE
    ControlOnEdge(CLK := IoDriver.ControlOnButton);
    ControlOffEdge(CLK := IoDriver.ControlOffButton);
END_IF
IF ControlOffEdge.Q THEN
    PneumaticPress.RequestLocalControl(ControlOn := FALSE);
ELSIF ControlOnEdge.Q THEN
    PneumaticPress.RequestLocalControl(ControlOn := TRUE);
END_IF
// Adopt the relay chain's established state: it is the authority. Without this
// the PLC can sit with no power request while K911_Y32 shows control is already
// ON (observed on the press), leaving PLC and hardware permanently out of step.
// One-shot: re-issuing POWER_ON every scan would re-fault the power group on
// any momentary permit dip and spam the event log. Latch on the feedback's
// rising edge only, and re-arm the latch when control drops away.
ControlOnAdopted(CLK := PowerHal.PowerFeedback);
IF NOT USE_SIMULATION AND ControlOnAdopted.Q AND NOT ControlOffEdge.Q THEN
    PneumaticPress.RequestLocalControl(ControlOn := TRUE);
END_IF

IF USE_SIMULATION THEN
    SimulationDriver.M_ReadInputs(DoorHal := DoorHal, TwoHandHal := TwoHandHal,
        PowerHal := PowerHal, PartPresentHal := PartPresentHal,
        AirPressureHal := AirPressureHal, RawEStopHealthy := RawEStopHealthy,
        SafeEStopOk := SafeEStopOk, SafeGuardClosed := SafeGuardClosed,
        SafeTwoHandActive := SafeTwoHandActive,
        SafePneumaticPermit := SafePneumaticPermit,
        SafetyFieldbusHealthy := SafetyFieldbusHealthy,
        StandardIoHealthy := StandardIoHealthy, SimEStopNc := SimEStopNc,
        SimLeftButton := SimLeftButton, SimRightButton := SimRightButton,
        SimSafetyValveOk := SimSafetyValveOk,
        SimFieldbusHealthy := SimFieldbusHealthy,
        SimPartPresent := SimPartPresent, SimAirPressureOk := SimAirPressureOk,
        PowerRequested := PowerHal.EnableRequestOut);
ELSE
    // The project Hardware Driver is the only raw process-image consumer.
    IoDriver.M_ReadInputs(PressHal := PressHal, DoorHal := DoorHal,
        SlideHal := SlideHal, TwoHandHal := TwoHandHal, PowerHal := PowerHal,
        PartPresentHal := PartPresentHal, AirPressureHal := AirPressureHal,
        RawEStopHealthy := RawEStopHealthy, SafeEStopOk := SafeEStopOk,
        SafeGuardClosed := SafeGuardClosed, SafeTwoHandActive := SafeTwoHandActive,
        SafePneumaticPermit := SafePneumaticPermit,
        SafetyFieldbusHealthy := SafetyFieldbusHealthy,
        StandardIoHealthy := StandardIoHealthy);
END_IF
TwoHandHal.SafeActive := SafeTwoHandActive;
TwoHandHal.FieldbusHealthy := SafetyFieldbusHealthy;
PowerHal.SafetyPermit := SafePneumaticPermit;
PowerHal.FieldbusHealthy := StandardIoHealthy;

ControlDomain.M_Update(SafeEStopOk := SafeEStopOk,
    SafeGuardClosed := SafeGuardClosed, SafeTwoHandActive := SafeTwoHandActive,
    SafePneumaticPermit := SafePneumaticPermit,
    SafetyFieldbusHealthy := SafetyFieldbusHealthy,
    StandardIoHealthy := StandardIoHealthy, RawEStopHealthy := RawEStopHealthy,
    PowerFeedback := PowerHal.PowerFeedback,
    PowerRequested := PowerHal.EnableRequestOut,
    TwoHandFieldbusHealthy := TwoHandHal.FieldbusHealthy);
PneumaticPress.ControlDomain := ControlDomain.Status;

// §2.7/§8.12 framework acceptance fixture. Simulation supplies explicit healthy
// synthetic controller/time probes; a real target stays conspicuously
// unavailable until its platform metrics and documented sync source are wired.
IF USE_SIMULATION THEN
    HealthCpuLoadPct := 25.0;
    HealthMemoryAvailableMb := UDINT#1024;
    HealthTimeSource := 'SIMULATED';
ELSE
    HealthCpuLoadPct := 0.0;
    HealthMemoryAvailableMb := UDINT#0;
    HealthTimeSource := 'UNCONFIGURED';
END_IF
HealthProbe.Cyclic(ExpectedCycleUs := 1000, ExternalTaskOverrun := FALSE,
    ControllerAvailable := USE_SIMULATION,
    CpuLoadPct := HealthCpuLoadPct,
    MemoryAvailableMb := HealthMemoryAvailableMb,
    IpcAvailable := FALSE, IpcTemperatureC := 0.0,
    FanHealthy := TRUE, StorageHealthPct := 100.0,
    FieldbusAvailable := TRUE, FieldbusMasterHealthy := StandardIoHealthy,
    LostFrameCount := 0, SlaveErrorCount := 0,
    DcAvailable := USE_SIMULATION, DcSynchronized := USE_SIMULATION,
    TimeAvailable := USE_SIMULATION, TimeSynchronized := USE_SIMULATION,
    TimeSource := HealthTimeSource,
    TimeOffsetUs := 0, LastSyncAt := F_Now());
IF HealthProbe.Health.TaskAvailable THEN
    PneumaticPress.SetSystemHealth(Input := HealthProbe.Health, ParCfg := HealthConfig);
ELSE
    ; // first monotonic sample has no prior scan from which to derive a period
END_IF

// First execute ordinary control, then apply a standard-PLC withdrawal layer.
// This is defense in depth only: the real safety system owns pneumatic removal.
PneumaticPress();
OutputAuthority.M_Apply(PressHal := PressHal, DoorHal := DoorHal,
    SlideHal := SlideHal, PowerFeedback := PowerHal.PowerFeedback,
    SafePneumaticPermit := SafePneumaticPermit,
    StandardIoHealthy := StandardIoHealthy,
    HazardousRamPermit := SafeGuardClosed AND SafeTwoHandActive);
IF USE_SIMULATION THEN
    // Never leave physical outputs energized while virtual commissioning.
    IoDriver.M_ClearOutputs();
    SimulationDriver.M_RefreshPlant();
ELSE
    LampsOn := PneumaticPress.TwoHand.OutImm.Armed
        AND ControlDomain.Status.ReadyForStart
        AND PneumaticPress.OutImm.PartPresent AND PneumaticPress.OutImm.AirPressureOk;
    IoDriver.M_WriteOutputs(PressHal := PressHal, DoorHal := DoorHal,
        SlideHal := SlideHal, PowerHal := PowerHal, LampsOn := LampsOn,
        ControlCircuitMappingConfirmed := CONTROL_CIRCUIT_MAPPING_CONFIRMED);
END_IF
// Node state comes from the real EtherCAT master. §10.5.1 is a diagnostic
// surface, so the master is scanned only while a client is watching the bus
// view: the HMI sets FieldbusViewActive when its fieldbus page is open (the same
// on-demand gating the read tiers already apply to the topology data itself).
IoDriver.M_RefreshFieldbus(BusViewActive := FieldbusViewActive);

END_PROGRAM

// ---- 00_System/FB_PressControlOnCircuit.TcPOU
// Hardware Control-On adapter for a machine whose safety is a HARDWIRED relay
// chain (Bosch/Nexeed N54 D2 "Control On", Pilz-style), NOT a TwinSAFE
// controller. The standard PLC is not a safety function here: the relay circuit
// remains the safety authority. This adapter only RECONSTRUCTS the read-only
// GVL_PressSafety-equivalent status the rest of the application expects, from the
// ordinary process-image inputs and the relay-chain Control On feedback, so the
// HMI and interlocks reflect the real machine instead of failing closed on
// unlinked TwinSAFE aliases.
//
// It produces status only (no safe outputs). The functional EnableControlOn /
// SwitchControlOn requests to the relay chain are driven by the existing power
// group -> FB_PressIoDriver.M_WriteOutputs path, gated by
// ControlCircuitMappingConfirmed until the electrical semantics are confirmed.
FUNCTION_BLOCK FB_PressControlOnCircuit
VAR_OUTPUT
    // Read-only mirrors, matching the six GVL_PressSafety aliases + the raw
    // E-stop mirror the driver forwards. TRUE = healthy/safe/present.
    RawEStopHealthy       : BOOL;
    SafeEStopOk           : BOOL;
    SafeGuardClosed       : BOOL;
    SafeTwoHandActive     : BOOL;
    SafePneumaticPermit   : BOOL;
    SafetyFieldbusHealthy : BOOL;
    StandardIoHealthy     : BOOL;

    // --- N54 D2 functional requests to the relay chain (not safety outputs) ---
    // EnableControlOn is a PERMISSIVE, not a command: per the standard it is set
    // at the start of the cycle from "bus OK and control-off not pressed", and
    // reset by the Main/Safety-Valve add-ons when compressed-air monitoring
    // errors. It must NOT wait for an operator power request, which is why the
    // control circuit could never be energized headless.
    EnableControlOn : BOOL;
    // SwitchControlOn is the BUTTON coil: TRUE for exactly two seconds on the
    // rising edge of the Control On button, however long the button is held, so
    // the guard doors have time to lock. Control Off has priority and cancels it.
    SwitchControlOn : BOOL;
    ControlOffSet   : BOOL;   // per the standard: NOT EnableControlOn
END_VAR
VAR
    _onEdge       : R_TRIG;
    _switchTimer  : TON;
    _switchActive : BOOL;
END_VAR

;

// Reconstruct the status mirrors from raw relay/sensor inputs. All inputs are
// ordinary (non-safety-rated) process-image values; the relay chain owns the
// actual safety function. Called once per scan by FB_PressIoDriver, the sole
// GVL_PressIO consumer.
METHOD M_Evaluate
VAR_INPUT
    EStopHealthyMirror : BOOL; // _000K910A: ordinary E-stop-healthy mirror
    DoorClosed         : BOOL; // _101B201A: guard-door closed sensor
    LeftButton         : BOOL; // _101S102: left two-hand raw button
    RightButton        : BOOL; // _101S101: right two-hand raw button
    ControlOnFeedback  : BOOL; // _000K911_Y32: relay-chain Control On established
    BusOk              : BOOL; // EtherCAT process image valid (link master OP state)
    ControlOnButton    : BOOL; // _000BS901: IsControlOnButtonPressed
    ControlOffButton   : BOOL; // _000BS902: IsControlOffButtonPressed
    AirPressureOk      : BOOL; // compressed-air monitoring OK (Main/Safety Valve)
END_VAR
// Fieldbus health: the standard and (functional) safety I/O share one EtherCAT
// segment on this machine, so both mirror the bus-valid signal.
StandardIoHealthy     := BusOk;
SafetyFieldbusHealthy := BusOk;

// E-stop: the ordinary healthy mirror gated by a valid process image. This is a
// diagnostic mirror of the relay-chain E-stop, not an evaluated safe result.
RawEStopHealthy := EStopHealthyMirror;
SafeEStopOk     := EStopHealthyMirror AND BusOk;

// Guard: the door-closed sensor. Plausibility (per N54 D2 Safety Door add-on) is
// enforced in the relay chain; here it is the single available door signal.
SafeGuardClosed := DoorClosed AND BusOk;

// Two-hand: functional (both raw buttons) with E-stop healthy. The safety-rated
// two-hand evaluation lives in the relay chain; this drives interlock/HMI only.
SafeTwoHandActive := LeftButton AND RightButton AND SafeEStopOk AND BusOk;

// Pneumatic permit: the relay-chain Control On feedback IS the enabled state.
// Per N54 D2 the Main/Safety Valve add-ons already reset EnableControlOn on a
// compressed-air error and the Safety Door add-on on a guard error, so the
// K911_Y32 feedback subsumes air + guard monitoring. Gate on E-stop for defense
// in depth (the air-pressure inputs are read separately by the air HAL).
SafePneumaticPermit := ControlOnFeedback AND SafeEStopOk;

// --- N54 D2 Control On add-on logic ---------------------------------------
// "EnableControlOn := BusOk AND NOT ControlOffButtonPressed", then reset by the
// Main/Safety-Valve add-ons on a compressed-air error. Guard doors deliberately
// do NOT gate it: the standard states the add-on still sets EnableControlOn (and
// briefly SwitchControlOn) while doors are open - the relay chain enforces the
// door condition.
EnableControlOn := BusOk AND NOT ControlOffButton AND AirPressureOk;
ControlOffSet   := NOT EnableControlOn;

// SwitchControlOn: exactly two seconds from the button's rising edge, cancelled
// immediately by Control Off (which has priority over Control On).
_onEdge(CLK := ControlOnButton);
IF ControlOffButton OR _switchTimer.Q THEN
    _switchActive := FALSE;
ELSIF _onEdge.Q AND EnableControlOn THEN
    _switchActive := TRUE;
END_IF
_switchTimer(IN := _switchActive, PT := T#2S);
SwitchControlOn := _switchActive;
END_METHOD

END_FUNCTION_BLOCK
